VAR_GLOBAL CONSTANT
	MAX_BUFFER_SIZE : UDINT := 1000;
END_VAR

(* stored: Version 1.1.0.1
   GVL GVL: Id {650ff06d-db32-42aa-abea-5d8b8128dc81} *)
